TYPE csp_transfer_accumulator_belt_phase_status_enum :
(		
	CSP_TRANSFER_ACCUMULATOR_BELT_STATUS_PHASE_START							:= 0,
	CSP_TRANSFER_ACCUMULATOR_BELT_STATUS_PHASE_DISABLE 							:= 10,
	CSP_TRANSFER_ACCUMULATOR_BELT_STATUS_PHASE_ENABLE 							:= 20,	
	CSP_TRANSFER_ACCUMULATOR_BELT_STATUS_PHASE_ENABLED 							:= 30,
	CSP_TRANSFER_ACCUMULATOR_BELT_STATUS_PHASE_CALCULATE_SLAVE_POSITION_REQUEST	:= 31,
	CSP_TRANSFER_ACCUMULATOR_BELT_STATUS_PHASE_CALCULATING_SLAVE_POSITION		:= 32,
	CSP_TRANSFER_ACCUMULATOR_BELT_STATUS_PHASE_REQUESTED						:= 33,
	CSP_TRANSFER_ACCUMULATOR_BELT_STATUS_PHASE_PHASING							:= 34,
	CSP_TRANSFER_ACCUMULATOR_BELT_STATUS_PHASE_PHASED							:= 35,
	CSP_TRANSFER_ACCUMULATOR_BELT_STATUS_PHASE_REDEFINE							:= 40,
	CSP_TRANSFER_ACCUMULATOR_BELT_STATUS_PHASE_REDEFINED						:= 50,
	CSP_TRANSFER_ACCUMULATOR_BELT_STATUS_PHASE_DONE 							:= 900,
	CSP_TRANSFER_ACCUMULATOR_BELT_STATUS_PHASE_ERROR 							:= 999
) := CSP_TRANSFER_ACCUMULATOR_BELT_STATUS_PHASE_START;
END_TYPE

(* stored: Version 1.1.0.1, ProductVersion 3.1.4024.3
   DUT csp_transfer_accumulator_belt_phase_status_enum: Id {bce2d2c7-72e2-4034-8cd6-264cd4c7ce4f} *)
